// TIA Portal V17 export
// export: Created 2023-02-13T11:16:32.5516496Z, ExportSetting WithDefaults, DisplayName Totally Integrated Automation Portal, DisplayVersion V17, DisplayName TIA Portal Openness, DisplayVersion V17, DisplayName TIA Portal Teamcenter Gateway, DisplayVersion V17, DisplayName TIA Portal Version Control Interface, DisplayVersion V17, DisplayName SINAMICS Startdrive Advanced, DisplayVersion V17, DisplayName SINAMICS Startdrive G130, G150, S120, S150, SINAMICS MV, S210, DisplayVersion V17, DisplayName SINAMICS Startdrive G110M, G120, G120C, G120D, G120P, G115D, DisplayVersion V17, DisplayName STEP 7 Professional, DisplayVersion V17, DisplayName STEP 7 Safety, DisplayVersion V17, DisplayName WinCC Professional, DisplayVersion V17
DATA_BLOCK "IO Analog Preparation_DB"   // DB13
VERSION : 0.1
// stored: AutoNumber true, DBAccessibleFromOPCUA true, DBAccessibleFromWebserver true, InstanceOfName IO Analog Preparation, InstanceOfType FB
"IO Analog Preparation"
   // VAR_INPUT
   //    Init : Bool;
   //    Reset : Bool;
   // END_VAR
   // VAR
   //    "LT-01.01" : "Ana_w_K1K2";
   //    "TT-01.01" : "Ana_w_K1K2";
   //    "TT-01.02" : "Ana_w_K1K2";
   //    "LT-02.01" : "Ana_w_K1K2";
   //    "LT-03.01" : "Ana_w_K1K2";
   //    "LT-04.01" : "Ana_w_K1K2";
   //    "LT-05.01" : "Ana_w_K1K2";
   //    "LT-06.01" : "Ana_w_K1K2";
   //    "LT-07.01" : "Ana_w_K1K2";
   //    "LT-08.01" : "Ana_w_K1K2";
   //    "LT-09.01" : "Ana_w_K1K2";
   //    "LT-10.01" : "Ana_w_K1K2";
   //    "TT-51.01" { S7_SetPoint := 'True'} : "Ana_w_K1K2";
   //    "CV-51.11" { S7_SetPoint := 'True'} : "Ana_w_K1K2";
   //    "FT-51.01" { S7_SetPoint := 'True'} : "Ana_w_K1K2";
   //    "FT-02.01" { S7_SetPoint := 'True'} : "Ana_w_K1K2";
   //    "FT-02.01Com" { S7_SetPoint := 'True'} : "Read FT Comm";
   //    "FT-03.01" { S7_SetPoint := 'True'} : "Ana_w_K1K2";
   //    "FT-03.01Com" { S7_SetPoint := 'True'} : "Read FT Comm";
   //    "FT-04.01" { S7_SetPoint := 'True'} : "Ana_w_K1K2";
   //    "FT-04.01Com" { S7_SetPoint := 'True'} : "Read FT Comm";
   //    "FT-05.01" { S7_SetPoint := 'True'} : "Ana_w_K1K2";
   //    "FT-05.01Com" { S7_SetPoint := 'True'} : "Read FT Comm";
   //    "FT-06.01" { S7_SetPoint := 'True'} : "Ana_w_K1K2";
   //    "FT-06.01Com" { S7_SetPoint := 'True'} : "Read FT Comm";
   //    "FT-07.01" { S7_SetPoint := 'True'} : "Ana_w_K1K2";
   //    "FT-07.01Com" { S7_SetPoint := 'True'} : "Read FT Comm";
   //    "FT-08.01" { S7_SetPoint := 'True'} : "Ana_w_K1K2";
   //    "FT-08.01Com" { S7_SetPoint := 'True'} : "Read FT Comm";
   //    "FT-09.01" { S7_SetPoint := 'True'} : "Ana_w_K1K2";
   //    "FT-09.01Com" { S7_SetPoint := 'True'} : "Read FT Comm";
   //    "FT-10.01" { S7_SetPoint := 'True'} : "Ana_w_K1K2";
   //    "FT-10.01Com" { S7_SetPoint := 'True'} : "Read FT Comm";
   // END_VAR
BEGIN
END_DATA_BLOCK
